FUNCTION_BLOCK AB_BYTE_TO_B (* Composite FB for convert AYTE to AB *)
  (* Standard: 61499-2; Description: Copyright (c) 2024 HR Agrartechnik GmbH This program and the accompanying materials are made available under the terms of the Eclipse Public License 2.0 which is available at https://www.eclipse.org/legal/epl-2.0/ SPDX-License-Identifier: EPL-2.0 *)
  (* Version 1.0, 2024-04-24, Franz Höpfinger, HR Agrartechnik GmbH *)
  PACKAGE adapter::conversion::unidirectional;
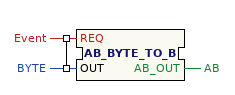
  EVENT_INPUT
    REQ WITH OUT; (* Request to Adapter *)
  END_EVENT
  VAR_INPUT
    OUT : BYTE; (* Output data to Adapter *)
  END_VAR
  PLUGS
    AB_OUT : adapter::types::unidirectional::AB; (* Adapter Output *)
  END_PLUGS
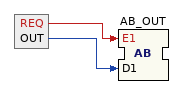
  EVENT_CONNECTIONS
    REQ TO AB_OUT.E1;
  END_CONNECTIONS
  DATA_CONNECTIONS
    OUT TO AB_OUT.D1;
  END_CONNECTIONS
END_FUNCTION_BLOCK
